FUNCTION_BLOCK PMLStateMachine IMPLEMENTS IPmlStateMachine
VAR_INPUT
END_VAR
VAR_OUTPUT
END_VAR
VAR
	_pmlStateMachine : Tc3_PackML_V2.PML_StateMachine;
	_pmlModeMachine : Tc3_PackML_V2.PML_UnitModeManager;
	_subUnits : ARRAY[0..9] OF IPmlStateMachine;
	subUnitArray : ARRAY[0..9] OF ST_PMLSubUnitInfo;
	_SubUnitReference: ST_PMLSubUnitInfoRef;
	modeChangeTrigger : Tc2_Standard.R_TRIG;
	i: DINT;
END_VAR

IF _SubUnitReference.NoOfSubUnits <> 0 THEN
	FOR i := 0 TO 9 DO
		IF _subUnits[i] <> 0 THEN
			subUnitArray[i].eState := _subUnits[i].GetCurrentState();
			subUnitArray[i].Active := True;
		END_IF
	END_FOR
	_SubUnitReference.pArray := ADR(subUnitArray);
	_SubUnitReference.ArraySize := SIZEOF(subUnitArray);
END_IF

_pmlStateMachine(eMode := _pmlModeMachine.eModeStatus, stSubUnitInfoRef := _SubUnitReference);
_pmlModeMachine(eState := _pmlStateMachine.eState, bExecute := modeChangeTrigger.Q);
modeChangeTrigger();

METHOD PUBLIC GetCurrentMode : E_PmlProtectedUnitMode
VAR_INPUT
END_VAR
GetCurrentMode := _pmlModeMachine.eModeStatus;
END_METHOD

METHOD PUBLIC GetCurrentState : E_PMLState
VAR_INPUT
END_VAR
GetCurrentState := _pmlStateMachine.eState;
END_METHOD

METHOD GetNumberOfSubUnits : INT
VAR_INPUT
END_VAR
END_METHOD

METHOD PUBLIC PmlModeCommand : Bool
VAR_INPUT
	Mode : E_PMLProtectedUnitMode;
END_VAR
_pmlModeMachine.eModeCommand := Mode;
modeChangeTrigger.CLK := true;
END_METHOD

METHOD PUBLIC PmlStateCommand : BOOL
VAR_INPUT
	Command : E_PMLCommand;
END_VAR
_pmlStateMachine.eCommand := Command;
END_METHOD

METHOD PUBLIC RegisterSubUnit : BOOL
VAR_INPUT
	SubUnit : IPmlStateMachine;
END_VAR
FOR i := 0 TO 9 DO
	IF _subUnits[i] = 0 THEN
		_subUnits[i] := SubUnit;
		_SubUnitReference.NoOfSubUnits := i + 1;
		EXIT;
	END_IF
END_FOR
END_METHOD

METHOD PUBLIC SetStateComplete : BOOL
VAR_INPUT
END_VAR
_pmlStateMachine.M_StateComplete();
END_METHOD

END_FUNCTION_BLOCK

(* stored: Version 1.1.0.1, ProductVersion 3.1.4024.11
   POU PMLStateMachine: Id {3acb0ffb-9e75-4713-9784-09cf44e02b1d}, SpecialFunc None
   Method GetCurrentMode: Id {a543b351-ed82-4c40-8e92-064ccf7f04ae}
   Method GetCurrentState: Id {fde5987d-e732-4f9a-a35a-61dbb1d8cf74}
   Method GetNumberOfSubUnits: Id {88b4d87a-c202-4a48-953a-5b41a16e252c}
   Method PmlModeCommand: Id {469ac633-6523-4ddf-8fdb-717cd972e2a4}
   Method PmlStateCommand: Id {21267235-cc94-44f6-b36d-074b99cb1582}
   Method RegisterSubUnit: Id {84da2a36-1704-4d61-bb15-d59bd2871aa6}
   Method SetStateComplete: Id {c21d0ca2-33a0-483f-96fc-a34e86036bc2} *)
